(* CODESYS project 01_SimpleFileWrite_csv.ecp

Project tree, tasks and I/O mapping:
  PFC200 : 750-8212 PFC200 G2 2ETH RS, WAGO, order no. 0750-8212, version 5.16.3.46
    application Application
      libraries: ; WagoAppFileDir, 1.6.2.1 (WAGO); WagoAppTime, 1.7.3.4 (WAGO)
      task PLC_Task (cyclic, interval 50 ms, priority 15) calls PLC_PRG
      program PLC_PRG [ST]
      data type typWriteData
    ProjectConfiguration
    Kbus : Kbus, WAGO, version 1.4.0.2
        unmapped channels: K-BUS diagnostics
    MODBUS
      MODBUS : MODBUS, WAGO, order no. n/a, version 1.1.1.16
    Serial
      COM1 : COM1, WAGO, version 0.0.0.19
    Common.PCI
    EtherNet/IP
      Ethernet : Ethernet, WAGO, version 35.16.0.0
          settings: IPAddress = [192, 168, 1, 212]; SubnetMask = [0, 0, 0, 0]; MACAddress = [16#00, 16#00, 16#00, 16#00, 16#00, 16#00]; NetworkInterfaceName = 'br0'; NetworkInterfaceName = "br0"
  00000000-0000-0000-0000-000000000000|C:\Users\u0100068\AppData\Local\Temp\c002284be6ff408abbc2a299aaf6497e\e868b832187f4f1a859da50215710801\Project.xml
*)

// PFC200/Application/typWriteData
{attribute 'qualified_only'}
{attribute 'strict'}
TYPE typWriteData :
(	// enumeration for the state machine
	eWaitForStart,
	eWriteData,
	eCloseFile,
	eErrorHandling
);
END_TYPE

// PFC200/Application/PLC_PRG
PROGRAM PLC_PRG
VAR
	fbWriteCsv:		WagoAppFileDir.FbSimpleWriteFile_cpt;
	xWriteData, xOpen, xIsOpen, xIsIdle, xError, xTrigger: BOOL;
	sName:			STRING(30) := '/var/www/myCSVfile.csv';	// call this file with your browser
	sSendString:	STRING(40);
	IResult:		FbResult;
	sDescription:	STRING;
	xResultError:	BOOL;
	iState:			typWriteData;
	stDateTime:		WagoTypes.typWagoTimeComponents;
	uiCount: UINT;
END_VAR

// get date and time from the controller as single variables
stDateTime := FuGetLocalTimeComponents();
// call the fb, remark: there's no "append to file", there's only "write file"
FbWriteCsv(
	xOpen		:= xOpen,
	xIsOpen		=> xIsOpen,
	xIsIdle		=> xIsIdle,
	xError		=> xError,
	xTrigger	:= xTrigger,
	oStatus		=> IResult,
	sName		:= sName,
	pTxBuffer	:= ADR(sSendString),
	udiTxNBytes	:= TO_UDINT(LEN(STR := sSendString)));
// get the feedback of the fb as string and as bool

sDescription := IResult.GetDescription();
xResultError := IResult.IsError();


// the state machine
CASE iState OF
	typWriteData.eWaitForStart:		// wait for the start bit
		// open the connection
		IF xWriteData THEN
			xOpen := TRUE;
		END_IF
		// if the connection is open, do something
		IF xIsOpen THEN
			uiCount:=uiCount+1;
			// define the send string with "format"
			sSendString := Format4(	sFormat := 'Dataset;%02i:%02i:%02i;%02i;$R$N ',
									p1		:= ADR(stDateTime.uiHour),
									p2		:= ADR(stDateTime.uiMinute),
									p3		:= ADR(stDateTime.uiSecond),
									p4		:= ADR(uiCount));
			// fire the trigger
			xTrigger := TRUE;
			// go to the next state
			iState := typWriteData.eWriteData;
		END_IF
	typWriteData.eWriteData:
		// if the trigger has been reset, the fb is ready
		IF NOT xTrigger THEN
			// close the connection
			xOpen := FALSE;
			iState := typWriteData.eCloseFile;
		END_IF
	typWriteData.eCloseFile:
		// wait for the connection being closed
		IF NOT xIsOpen THEN
			xWriteData := FALSE;
			iState := typWriteData.eWaitForStart;
		END_IF
	typWriteData.eErrorHandling:
		uiCount:=0;
				// - ...tbd
END_CASE;

END_PROGRAM
